FUNCTION_BLOCK FB_CreateTepletate2 EXTENDS FB_Base IMPLEMENTS ITF_BaseCreateTemplateOfRecipe
VAR
END_VAR

METHOD CreateTamplateOfRecipe : BOOL
VAR_INPUT
	itfRecipe				: ITF_BaseCreatingTemplateMethod;	//interfejs do obsługi receptur
END_VAR
VAR
	sttmpSkladnik			: ST_BaseDescriptor;
	uiNumberOfTeplates		: UINT;
END_VAR
THIS^.SetText (eLocation := E_BaseLocation.pl, wsDescription := "Nazwa szablonu 2 PL");
THIS^.SetText (eLocation := E_BaseLocation.en, wsDescription := "Nazwa szablonu 2 EN");
THIS^.SetText (eLocation := E_BaseLocation.de, wsDescription := "Nazwa szablonu 2 DE");
itfRecipe.AddTemplate (stTexts	:= GVL.fbRecipe.GetTexts ());
uiNumberOfTeplates	:= itfRecipe.GetNumberOfTemplate ();

THIS^.SetTextIn (stIN := sttmpSkladnik, eLocation := E_BaseLocation.pl, wsDescription := "Nazwa skladnika 1 PL");
THIS^.SetTextIn (stIN := sttmpSkladnik, eLocation := E_BaseLocation.en, wsDescription := "Nazwa skladnika 1 EN");
THIS^.SetTextIn (stIN := sttmpSkladnik, eLocation := E_BaseLocation.de, wsDescription := "Nazwa skladnika 1 DE");
THIS^.SetMaxIn (stIN := sttmpSkladnik, rMax := 10000);
THIS^.SetMinIn (stIN := sttmpSkladnik, rMin := 1);
THIS^.SetValueIn (stIN := sttmpSkladnik, rValue := 1111);
THIS^.SetDefaultValueIn (stIN := sttmpSkladnik, rDefaultValue := 1111);
THIS^.SetUnitIn (stIN := sttmpSkladnik, sUnit := 'mm');
itfRecipe.AddIngredientToTemplate (uiNumber := uiNumberOfTeplates, stIngredient := sttmpSkladnik);
END_METHOD

END_FUNCTION_BLOCK

(* stored: Version 1.1.0.1, ProductVersion 3.1.4024.15
   POU FB_CreateTepletate2: Id {33a5c29b-21b8-4f84-a2c3-53bed86efa1f}, SpecialFunc None
   Method CreateTamplateOfRecipe: Id {2f2fc05b-80ed-4202-b089-6c118e05dafa} *)
